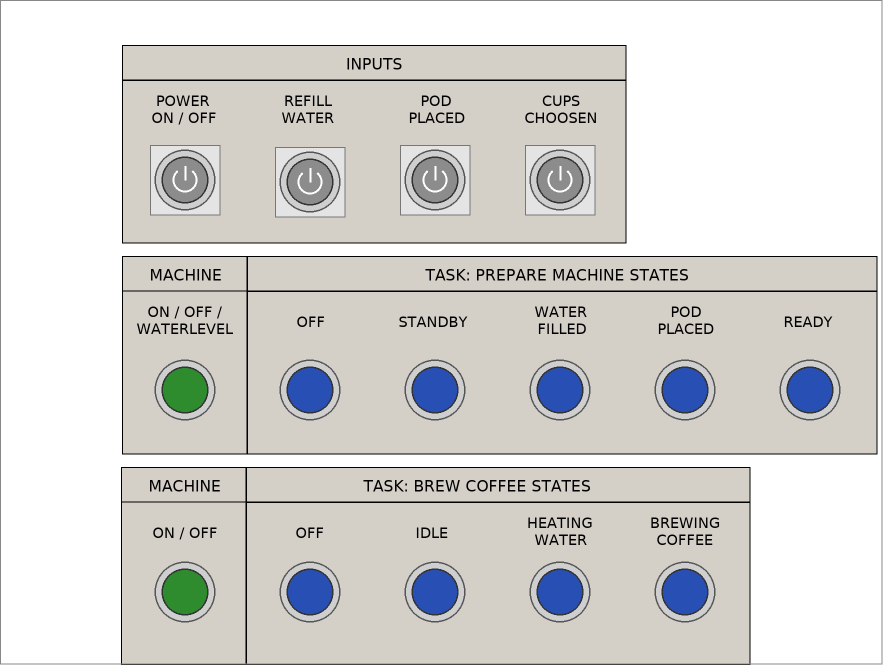
VISUALIZATION Process  // 883x665
    Rectangle (247,291 630x163)
    Rectangle (247,256 630x35)
    Rectangle (122,256 125x198)
    Label (358,307 150x30), "STANDBY"
    Label (236,307 150x30), "OFF"
    Label (486,297 150x30), "WATER"
    Label (611,297 150x30), "POD"
    Rectangle (122,256 125x35)
    Label (111,260 150x30), "MACHINE"
    Label (487,314 150x30), "FILLED"
    Label (611,314 150x30), "PLACED"
    Label (395,260 325x30), "TASK: PREPARE MACHINE STATES"
    Rectangle (246,502 504x163)
    Rectangle (246,467 504x35)
    Rectangle (121,467 125x198)
    Lamp1 (150,355 70x70), variable: PrepareMachine.LED, style: Lamp-Lamp1-Green
    Lamp1 (275,355 70x70), variable: PrepareMachine.OFF, style: Lamp-Lamp1-Blue
    Lamp1 (400,355 70x70), variable: PrepareMachine.Standby, style: Lamp-Lamp1-Blue
    Lamp1 (525,355 70x70), variable: PrepareMachine.WaterFilled, style: Lamp-Lamp1-Blue
    Lamp1 (650,355 70x70), variable: PrepareMachine.PodPlaced, style: Lamp-Lamp1-Blue
    Lamp1 (775,355 70x70), variable: PrepareMachine.Ready, style: Lamp-Lamp1-Blue
    Label (110,518 150x30), "ON / OFF"
    Label (357,518 150x30), "IDLE"
    Label (235,518 150x30), "OFF"
    Label (485,508 150x30), "HEATING"
    Label (610,508 150x30), "BREWING"
    Lamp1 (650,557 70x70), variable: BrewCoffee.BrewCoffee, style: Lamp-Lamp1-Blue
    Lamp1 (525,557 70x70), variable: BrewCoffee.HeatingWater, style: Lamp-Lamp1-Blue
    Lamp1 (400,557 70x70), variable: BrewCoffee.Idle, style: Lamp-Lamp1-Blue
    Lamp1 (275,557 70x70), variable: BrewCoffee.OFF, style: Lamp-Lamp1-Blue
    Lamp1 (150,557 70x70), variable: BrewCoffee.LED, style: Lamp-Lamp1-Green
    Rectangle (121,467 125x35)
    Label (110,471 150x30), "MACHINE"
    Label (486,525 150x30), "WATER"
    Label (610,525 150x30), "COFFEE"
    Label (347,471 261x30), "TASK: BREW COFFEE STATES"
    Label (110,297 150x30), "ON / OFF /"
    Label (110,314 150x30), "WATERLEVEL"
    Label (733,307 150x30), "READY"
    Rectangle (122,80 504x163)
    Rectangle (122,45 504x35)
    Label (361,86 150x30), "POD"
    Label (486,86 150x30), "CUPS"
    Label (362,103 150x30), "PLACED"
    Label (486,103 150x30), "CHOOSEN"
    Label (244,49 261x30), "INPUTS"
    Label (108,86 150x30), "POWER"
    Label (233,86 150x30), "REFILL"
    Label (109,103 150x30), "ON / OFF"
    Label (233,103 150x30), "WATER"
    PowerSwitch (150,145 70x70), variable: GVL.Power, behaviour: TOGGLE, style: Switch-PowerSwitch-Gray
    PowerSwitch (400,145 70x70), variable: PrepareMachine.Pod, behaviour: TOGGLE, style: Switch-PowerSwitch-Gray
    PowerSwitch (525,145 70x70), variable: PrepareMachine.CupsChoosen, behaviour: TOGGLE, style: Switch-PowerSwitch-Gray
    PowerSwitch (275,147 70x70), variable: PrepareMachine.WaterRefilled, behaviour: TOGGLE, style: Switch-PowerSwitch-Gray
END_VISUALIZATION

(* stored: Version 1.1.0.1, ProductVersion 3.1.4024.12
   Visu Process: Id {299d2d01-938e-459d-bbaa-a0a16e3cee39} *)
